Fanuc KAREL source: wcntspeedup.kl

PROGRAM wcntspeedup
%NOLOCKGROUP
VAR
  p : POSITION
  q : POSITION
  i : INTEGER
  r : REAL
BEGIN
  WITH $CNT_SPEEDUP = TRUE MOVE TO p
END wcntspeedup
